(* Logix 5000 project; controller ARS14002_PLC vendor 1 type 14 code 218 rev 30.11; software revision 30.01; part 12 of 13 *)
(* tags used below, declared in another part *)
   AN_1000C : CM_AI_SCL;
   AN_200A : CM_AI_SCL;
   ARS_COLLECT : BOOL;
   ARS_FULL_COLLECTION : BOOL;
   ARS_FULL_COLLECTION_LATCH : BOOL;   // LATCHES THE FIRST TIME ARS HITS FULL COLLECTION DURING A MODE_ATOMIZE
   ARS_FULL_COLLECTION_TMR : TIMER;
   AT2_AtomizingStatus_OSF_OB : BOOL;
   AT2_FT_202_TOTAL_HEAT : REAL;
   AT2_HIBON_DISCHARGE_TEMP : REAL;
   AT2_HIBON_DISCHARGE_TEMP_MAX : REAL;
   AT2_PLANT_ATOMIZING : BOOL;
   AT2_PLANT_COLLECTION_PERCENT : REAL;
   AT2_PLANT_COLLECTION_PERCENT_GOOD_GAS : REAL;
   AT2_PLANT_COLLECTION_TIME : TIMER;
   AT2_PLANT_GOOD_GAS_PERCENT : REAL;
   AT2_PLANT_GOOD_GAS_TIME : TIMER;   // AT2 total time with good gas and no collection stops
   AT2_PLANT_GOOD_H2O_PERCENT : REAL;
   AT2_PLANT_GOOD_H2O_TIME : TIMER;   // AT2 time with good dew point and no collection stop
   AT2_PLANT_GOOD_O2_PERCENT : REAL;
   AT2_PLANT_GOOD_O2_TIME : TIMER;   // AT2 time with good O2 and no collection stop
   AT2_PLANT_LIKELY_COLLECTION_TIME : TIMER;
   AT2_PLANT_MAX_H2O : REAL;
   AT2_PLANT_MAX_O2 : REAL;
   AT2_PLANT_POST_HEAT_NOTIFICATION_TON : TIMER;
   AT2_V1_OPEN : BOOL;
   AT2_V1_OPEN_OSR_OB : BOOL;
   AT2_V1_OPEN_OSR_SB : BOOL;
   AT2_V1_OPEN_POSTHEAT_CTR : COUNTER;
   AT3_AtomizingStatus_OSF_OB : BOOL;
   AT3_FT_202_TOTAL_HEAT : REAL;
   AT3_HIBON_DISCHARGE_TEMP : REAL;
   AT3_HIBON_DISCHARGE_TEMP_MAX : REAL;
   AT3_PLANT_ATOMIZING : BOOL;
   AT3_PLANT_COLLECTION_PERCENT : REAL;
   AT3_PLANT_COLLECTION_PERCENT_GOOD_GAS : REAL;
   AT3_PLANT_COLLECTION_TIME : TIMER;
   AT3_PLANT_GOOD_GAS_PERCENT : REAL;
   AT3_PLANT_GOOD_GAS_TIME : TIMER;   // total time with good gas and no collection stops
   AT3_PLANT_GOOD_H2O_PERCENT : REAL;
   AT3_PLANT_GOOD_H2O_TIME : TIMER;   // time with good dew point and no collection stop
   AT3_PLANT_GOOD_O2_PERCENT : REAL;
   AT3_PLANT_GOOD_O2_TIME : TIMER;   // time with good O2 and no collection stop
   AT3_PLANT_LIKELY_COLLECTION_TIME : TIMER;
   AT3_PLANT_MAX_H2O : REAL;
   AT3_PLANT_MAX_O2 : REAL;
   AT3_PLANT_POST_HEAT_NOTIFICATION_TON : TIMER;
   AT3_V1_OPEN : BOOL;
   AT3_V1_OPEN_OSR_OB : BOOL;
   AT3_V1_OPEN_OSR_SB : BOOL;
   AT3_V1_OPEN_POSTHEAT_CTR : COUNTER;
   CALC_FT_1002_MONTH_RETURN : REAL;
   CALC_FT_1002_MONTH_TOTALIZER_RESET : BOOL;
   CALC_FT_1002_MONTH_TOTALIZER_START : BOOL;
   CALC_FT_1002_MONTH_TOTALIZER_STOP : BOOL;
   CALC_FT_1002_TOTAL_RETURN : REAL;
   CALC_FT_202_MONTH : REAL;
   CALC_FT_202_TOTAL_HEAT : REAL;
   CALC_NEXT_DAY_OSR_OB : BOOL;
   CALC_NEXT_MONTH_OSR_OB : BOOL;
   COLDBOX_REACTION_TMR : TIMER;
   COLDBOX_REACTION_TMR_SEC : REAL;
   FCV_1001 : CM_AO_VLV;
   FCV_1002 : CM_AO_VLV;
   FCV_101A : CM_AO_VLV;
   FCV_101A_ZT_OSR : BOOL;
   FCV_101B : CM_AO_VLV;
   FCV_101B_ZT_OSR : BOOL;
   FCV_101C : CM_AO_VLV;
   FCV_101C_ZT_OSR : BOOL;
   FCV_102A : CM_AO_VLV;
   FCV_102A_COLLECTION_CV_HIGH : REAL;
   FCV_102B : CM_AO_VLV;
   FCV_102B_COLLECTION_CV_HIGH : REAL;
   FCV_102C : CM_AO_VLV;
   FCV_102C_COLLECTION_CV_HIGH : REAL;
   FCV_1221 : CM_AO_VLV;
   FCV_1251 : CM_AO_VLV;
   FCV_202 : CM_AO_VLV;
   FCV_202_COLLECTION_CV_LOW : REAL;
   FCV_202_HEAT_AVG : REAL;
   FCV_202_HEAT_AVG_TON : TIMER;
   FCV_202_HEAT_TOTAL : REAL;
   FCV_202_SAMPLES : COUNTER;
   FCV_204 : CM_AO_VLV;
   FCV_204_COLLECTION_CV_HIGH : REAL;
   FCV_204_HEAT_AVG : REAL;
   FCV_204_HEAT_TOTAL : REAL;
   FCV_207 : CM_AO_VLV;
   FCV_504 : CM_AO_VLV;
   FCV_603 : CM_AO_VLV;
   FCV_605 : CM_AO_VLV;
   FCV_753 : CM_AO_VLV;
   FCV_754 : CM_AO_VLV;
   FCV_755 : CM_AO_VLV;
   FT_1002 : CM_AI_SCL;
   FT_202_ALT_SCFM : REAL;
   FULL_COLLECT_INTERRUPT_ALM : BOOL;
   FULL_COLLECT_INTERRUPT_ALM_TIME : DINT;
   FULL_COLLECT_INTERRUPT_ALM_TMR : TIMER;
   FULL_COLLECT_START_ALM : BOOL;
   FULL_COLLECT_START_ALM_TIME : DINT;
   FULL_COLLECT_START_ALM_TMR : TIMER;
   Heat_Counter_AT2 : DINT;
   Heat_Counter_AT3 : REAL;
   Heat_Counter_Month : REAL;
   Heat_Counter_Pilot : REAL;
   HEAT_TIMER_AT2 : TIMER;
   HEAT_TIMER_AT3 : TIMER;
   MODE_ATOMIZE : BOOL;
   P_800A_CAVIT_CTR_MONTH : COUNTER;
   P_800B_CAVIT_CTR_MONTH : COUNTER;
   P_800C_CAVIT_CTR_MONTH : COUNTER;
   P_800D_CAVIT_CTR_MONTH : COUNTER;
   Pilot_AtomizingStatus_OSF_OB : BOOL;
   PILOT_FT_202_TOTAL_HEAT : REAL;
   PILOT_PLANT_ATOMIZING : BOOL;
   PILOT_PLANT_MAX_H2O : REAL;
   PILOT_PLANT_MAX_O2 : REAL;
   PILOT_PLANT_POST_HEAT_NOTIFICATION_TON : TIMER;
   PWHMI_AtomizingStatus_OSR_OB : BOOL;
   SEND_AT2_PLANT_NOTICE : BOOL;
   SEND_AT3_PLANT_NOTICE : BOOL;
   SEND_PILOT_PLANT_NOTICE : BOOL;
   SV_202F : CM_DO_GENERIC;
   SV_802AX : CM_DO_GENERIC;
   SV_802AX_ONS : BOOL;
   SV_802BX : CM_DO_GENERIC;
   SV_802BX_ONS : BOOL;
   SV_802CX : CM_DO_GENERIC;
   SV_802CX_ONS : BOOL;
   SV_802DX : CM_DO_GENERIC;
   SV_802DX_ONS : BOOL;
   XV_802_VENT_COUNTER : COUNTER;
   XV_802_VENT_TOTAL_TIME : TIMER;
   ZT_1001 : CM_AI_SCL;
   ZT_1002 : CM_AI_SCL;
   ZT_101A : CM_AI_SCL;
   ZT_101B : CM_AI_SCL;
   ZT_101C : CM_AI_SCL;
   ZT_102A : CM_AI_SCL;
   ZT_102B : CM_AI_SCL;
   ZT_102C : CM_AI_SCL;
   ZT_1221 : CM_AI_SCL;
   ZT_1251 : CM_AI_SCL;
   ZT_202 : CM_AI_SCL;
   ZT_204 : CM_AI_SCL;
   ZT_207 : CM_AI_SCL;
   ZT_504 : CM_AI_SCL;
   ZT_603 : CM_AI_SCL;
   ZT_605 : CM_AI_SCL;
   ZT_753 : CM_AI_SCL;
   ZT_754 : CM_AI_SCL;
   ZT_755 : CM_AI_SCL;
(* MainProgram, continued *)

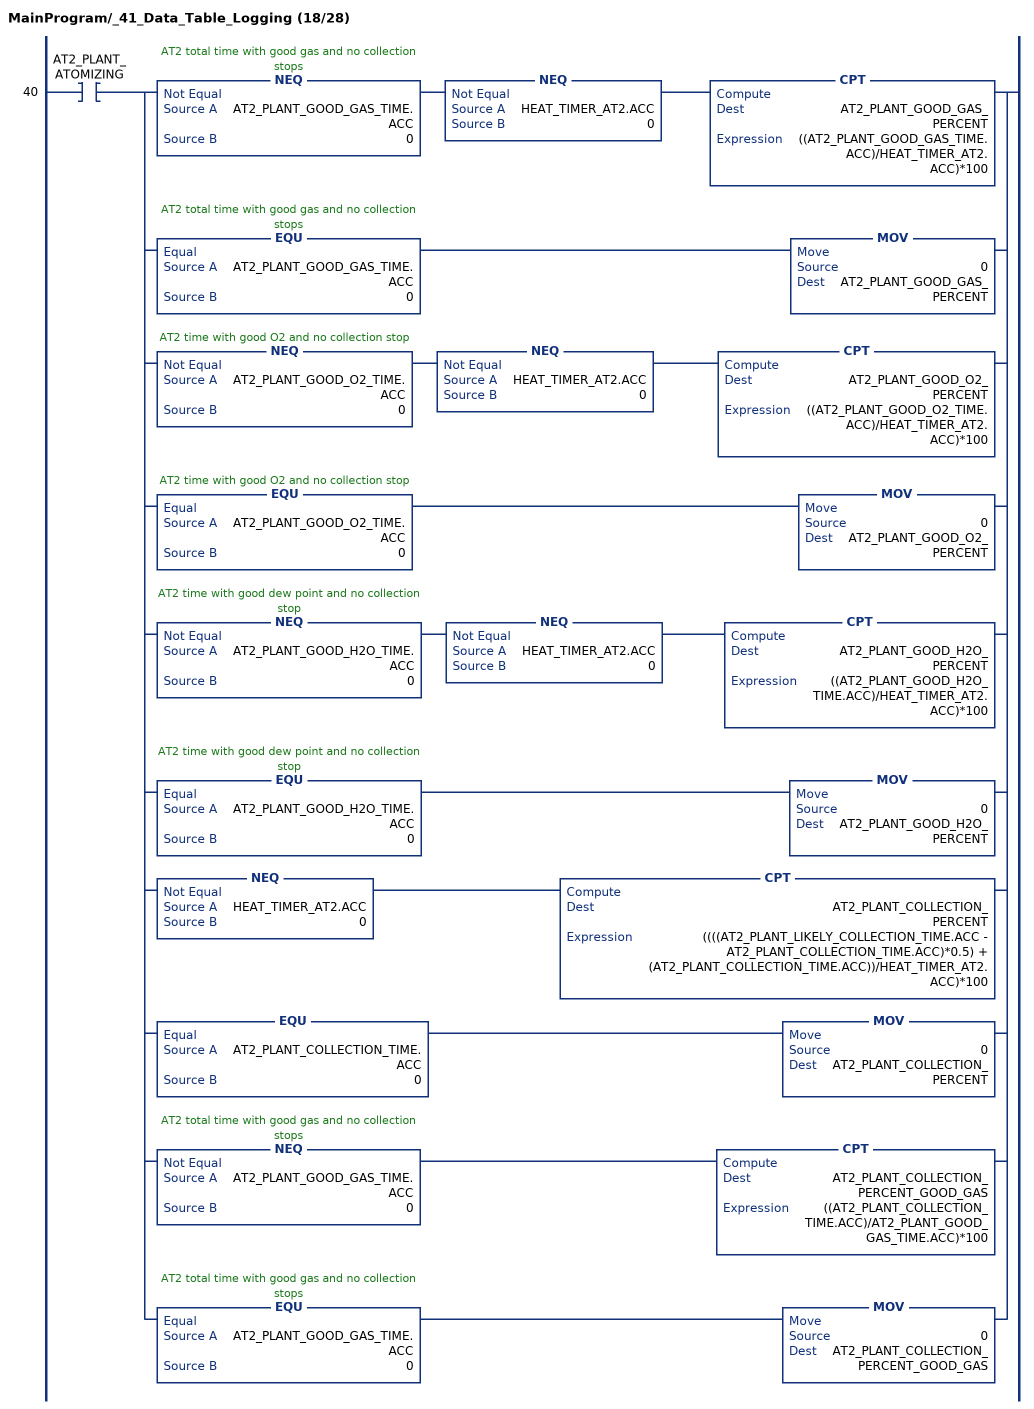
   [picture p246: MainProgram/_41_Data_Table_Logging rungs 40-40]
   40: XIC(AT2_PLANT_ATOMIZING)[NEQ(AT2_PLANT_GOOD_GAS_TIME.ACC,0) NEQ(HEAT_TIMER_AT2.ACC,0) CPT(AT2_PLANT_GOOD_GAS_PERCENT,((AT2_PLANT_GOOD_GAS_TIME.ACC)/HEAT_TIMER_AT2.ACC)*100) ,EQU(AT2_PLANT_GOOD_GAS_TIME.ACC,0) MOV(0,AT2_PLANT_GOOD_GAS_PERCENT) ,NEQ(AT2_PLANT_GOOD_O2_TIME.ACC,0) NEQ(HEAT_TIMER_AT2.ACC,0) CPT(AT2_PLANT_GOOD_O2_PERCENT,((AT2_PLANT_GOOD_O2_TIME.ACC)/HEAT_TIMER_AT2.ACC)*100) ,EQU(AT2_PLANT_GOOD_O2_TIME.ACC,0) MOV(0,AT2_PLANT_GOOD_O2_PERCENT) ,NEQ(AT2_PLANT_GOOD_H2O_TIME.ACC,0) NEQ(HEAT_TIMER_AT2.ACC,0) CPT(AT2_PLANT_GOOD_H2O_PERCENT,((AT2_PLANT_GOOD_H2O_TIME.ACC)/HEAT_TIMER_AT2.ACC)*100) ,EQU(AT2_PLANT_GOOD_H2O_TIME.ACC,0) MOV(0,AT2_PLANT_GOOD_H2O_PERCENT) ,NEQ(HEAT_TIMER_AT2.ACC,0) CPT(AT2_PLANT_COLLECTION_PERCENT,((((AT2_PLANT_LIKELY_COLLECTION_TIME.ACC - AT2_PLANT_COLLECTION_TIME.ACC)*0.5) + (AT2_PLANT_COLLECTION_TIME.ACC))/HEAT_TIMER_AT2.ACC)*100) ,EQU(AT2_PLANT_COLLECTION_TIME.ACC,0) MOV(0,AT2_PLANT_COLLECTION_PERCENT) ,NEQ(AT2_PLANT_GOOD_GAS_TIME.ACC,0) CPT(AT2_PLANT_COLLECTION_PERCENT_GOOD_GAS,((AT2_PLANT_COLLECTION_TIME.ACC)/AT2_PLANT_GOOD_GAS_TIME.ACC)*100) ,EQU(AT2_PLANT_GOOD_GAS_TIME.ACC,0) MOV(0,AT2_PLANT_COLLECTION_PERCENT_GOOD_GAS) ];
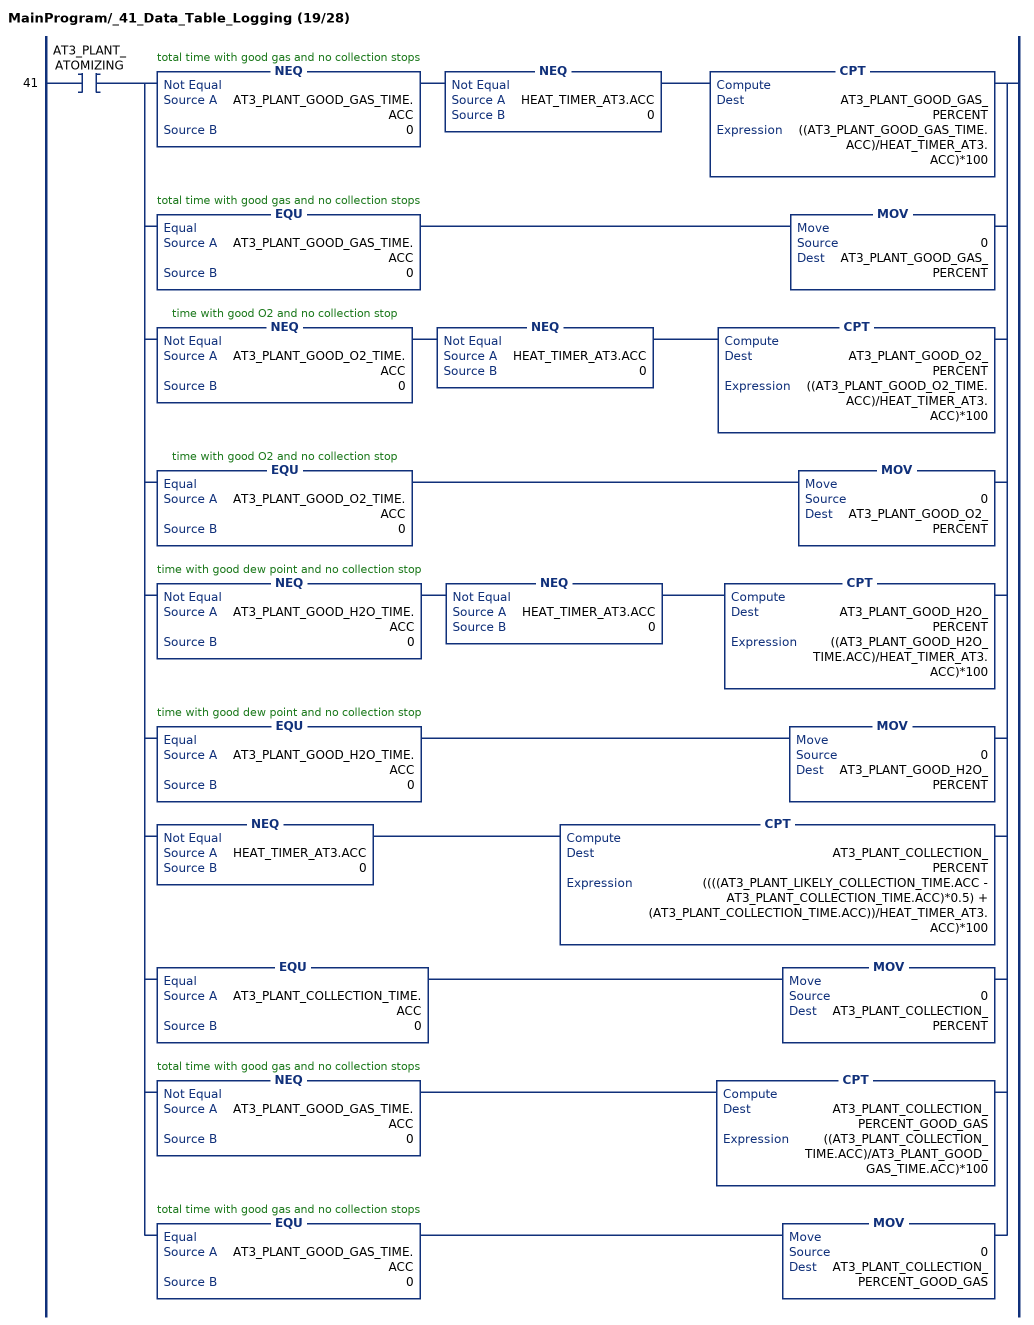
   41: XIC(AT3_PLANT_ATOMIZING)[NEQ(AT3_PLANT_GOOD_GAS_TIME.ACC,0) NEQ(HEAT_TIMER_AT3.ACC,0) CPT(AT3_PLANT_GOOD_GAS_PERCENT,((AT3_PLANT_GOOD_GAS_TIME.ACC)/HEAT_TIMER_AT3.ACC)*100) ,EQU(AT3_PLANT_GOOD_GAS_TIME.ACC,0) MOV(0,AT3_PLANT_GOOD_GAS_PERCENT) ,NEQ(AT3_PLANT_GOOD_O2_TIME.ACC,0) NEQ(HEAT_TIMER_AT3.ACC,0) CPT(AT3_PLANT_GOOD_O2_PERCENT,((AT3_PLANT_GOOD_O2_TIME.ACC)/HEAT_TIMER_AT3.ACC)*100) ,EQU(AT3_PLANT_GOOD_O2_TIME.ACC,0) MOV(0,AT3_PLANT_GOOD_O2_PERCENT) ,NEQ(AT3_PLANT_GOOD_H2O_TIME.ACC,0) NEQ(HEAT_TIMER_AT3.ACC,0) CPT(AT3_PLANT_GOOD_H2O_PERCENT,((AT3_PLANT_GOOD_H2O_TIME.ACC)/HEAT_TIMER_AT3.ACC)*100) ,EQU(AT3_PLANT_GOOD_H2O_TIME.ACC,0) MOV(0,AT3_PLANT_GOOD_H2O_PERCENT) ,NEQ(HEAT_TIMER_AT3.ACC,0) CPT(AT3_PLANT_COLLECTION_PERCENT,((((AT3_PLANT_LIKELY_COLLECTION_TIME.ACC - AT3_PLANT_COLLECTION_TIME.ACC)*0.5) + (AT3_PLANT_COLLECTION_TIME.ACC))/HEAT_TIMER_AT3.ACC)*100) ,EQU(AT3_PLANT_COLLECTION_TIME.ACC,0) MOV(0,AT3_PLANT_COLLECTION_PERCENT) ,NEQ(AT3_PLANT_GOOD_GAS_TIME.ACC,0) CPT(AT3_PLANT_COLLECTION_PERCENT_GOOD_GAS,((AT3_PLANT_COLLECTION_TIME.ACC)/AT3_PLANT_GOOD_GAS_TIME.ACC)*100) ,EQU(AT3_PLANT_GOOD_GAS_TIME.ACC,0) MOV(0,AT3_PLANT_COLLECTION_PERCENT_GOOD_GAS) ];
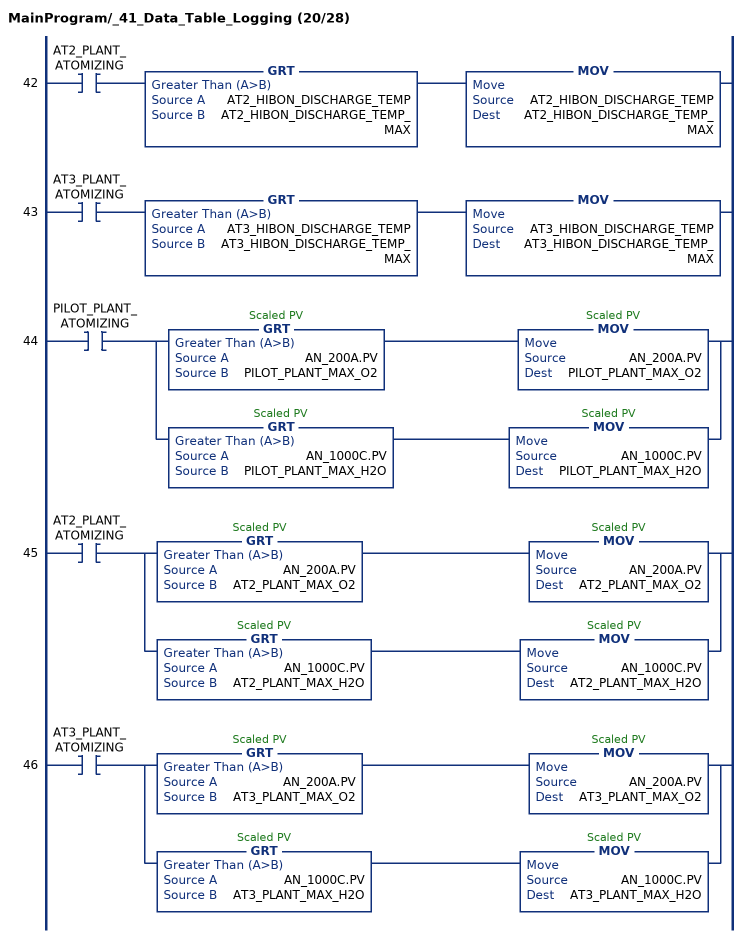
   42: XIC(AT2_PLANT_ATOMIZING)GRT(AT2_HIBON_DISCHARGE_TEMP,AT2_HIBON_DISCHARGE_TEMP_MAX)MOV(AT2_HIBON_DISCHARGE_TEMP,AT2_HIBON_DISCHARGE_TEMP_MAX);
   43: XIC(AT3_PLANT_ATOMIZING)GRT(AT3_HIBON_DISCHARGE_TEMP,AT3_HIBON_DISCHARGE_TEMP_MAX)MOV(AT3_HIBON_DISCHARGE_TEMP,AT3_HIBON_DISCHARGE_TEMP_MAX);
   44: XIC(PILOT_PLANT_ATOMIZING)[GRT(AN_200A.PV,PILOT_PLANT_MAX_O2) MOV(AN_200A.PV,PILOT_PLANT_MAX_O2) ,GRT(AN_1000C.PV,PILOT_PLANT_MAX_H2O) MOV(AN_1000C.PV,PILOT_PLANT_MAX_H2O) ];
   45: XIC(AT2_PLANT_ATOMIZING)[GRT(AN_200A.PV,AT2_PLANT_MAX_O2) MOV(AN_200A.PV,AT2_PLANT_MAX_O2) ,GRT(AN_1000C.PV,AT2_PLANT_MAX_H2O) MOV(AN_1000C.PV,AT2_PLANT_MAX_H2O) ];
   46: XIC(AT3_PLANT_ATOMIZING)[GRT(AN_200A.PV,AT3_PLANT_MAX_O2) MOV(AN_200A.PV,AT3_PLANT_MAX_O2) ,GRT(AN_1000C.PV,AT3_PLANT_MAX_H2O) MOV(AN_1000C.PV,AT3_PLANT_MAX_H2O) ];
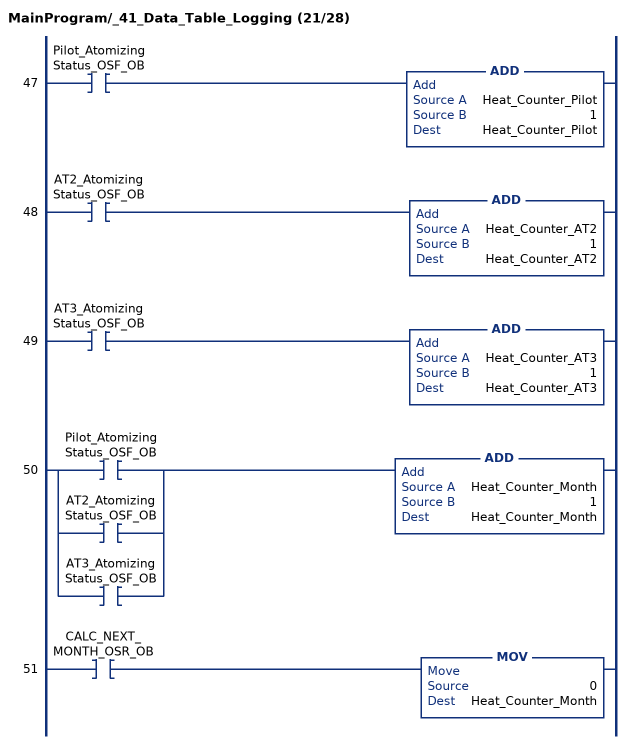
   47: XIC(Pilot_AtomizingStatus_OSF_OB)ADD(Heat_Counter_Pilot,1,Heat_Counter_Pilot);
   48: XIC(AT2_AtomizingStatus_OSF_OB)ADD(Heat_Counter_AT2,1,Heat_Counter_AT2);
   49: XIC(AT3_AtomizingStatus_OSF_OB)ADD(Heat_Counter_AT3,1,Heat_Counter_AT3);
   50: [XIC(Pilot_AtomizingStatus_OSF_OB) ,XIC(AT2_AtomizingStatus_OSF_OB) ,XIC(AT3_AtomizingStatus_OSF_OB) ]ADD(Heat_Counter_Month,1,Heat_Counter_Month);
   51: XIC(CALC_NEXT_MONTH_OSR_OB)MOV(0,Heat_Counter_Month);
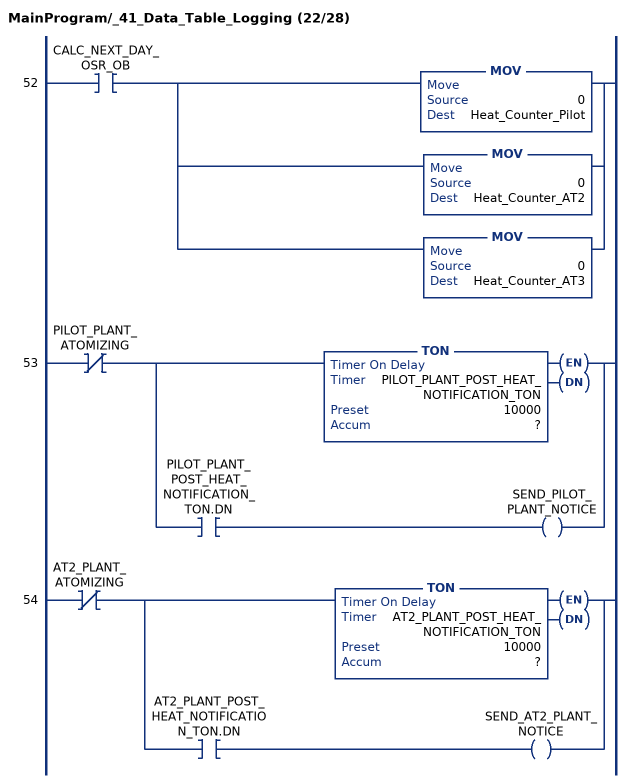
   52: XIC(CALC_NEXT_DAY_OSR_OB)[MOV(0,Heat_Counter_Pilot) ,MOV(0,Heat_Counter_AT2) ,MOV(0,Heat_Counter_AT3) ];
   53: XIO(PILOT_PLANT_ATOMIZING)[TON(PILOT_PLANT_POST_HEAT_NOTIFICATION_TON,?,?) ,XIC(PILOT_PLANT_POST_HEAT_NOTIFICATION_TON.DN) OTE(SEND_PILOT_PLANT_NOTICE) ];
   54: XIO(AT2_PLANT_ATOMIZING)[TON(AT2_PLANT_POST_HEAT_NOTIFICATION_TON,?,?) ,XIC(AT2_PLANT_POST_HEAT_NOTIFICATION_TON.DN) OTE(SEND_AT2_PLANT_NOTICE) ];
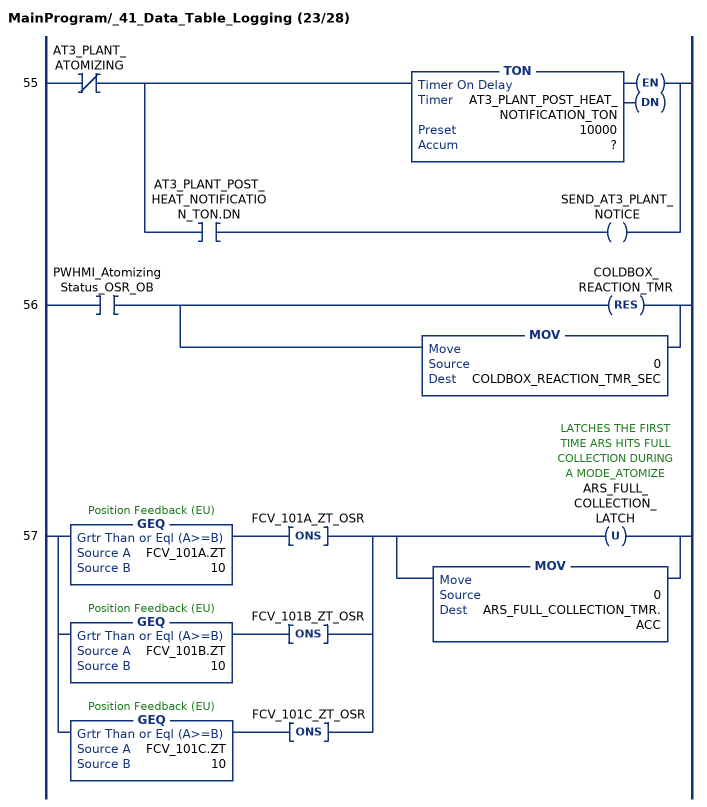
   55: XIO(AT3_PLANT_ATOMIZING)[TON(AT3_PLANT_POST_HEAT_NOTIFICATION_TON,?,?) ,XIC(AT3_PLANT_POST_HEAT_NOTIFICATION_TON.DN) OTE(SEND_AT3_PLANT_NOTICE) ];
   56: XIC(PWHMI_AtomizingStatus_OSR_OB)[RES(COLDBOX_REACTION_TMR) ,MOV(0,COLDBOX_REACTION_TMR_SEC) ];
   57: [GEQ(FCV_101A.ZT,10) ONS(FCV_101A_ZT_OSR) ,GEQ(FCV_101B.ZT,10) ONS(FCV_101B_ZT_OSR) ,GEQ(FCV_101C.ZT,10) ONS(FCV_101C_ZT_OSR) ][OTU(ARS_FULL_COLLECTION_LATCH) ,MOV(0,ARS_FULL_COLLECTION_TMR.ACC) ];
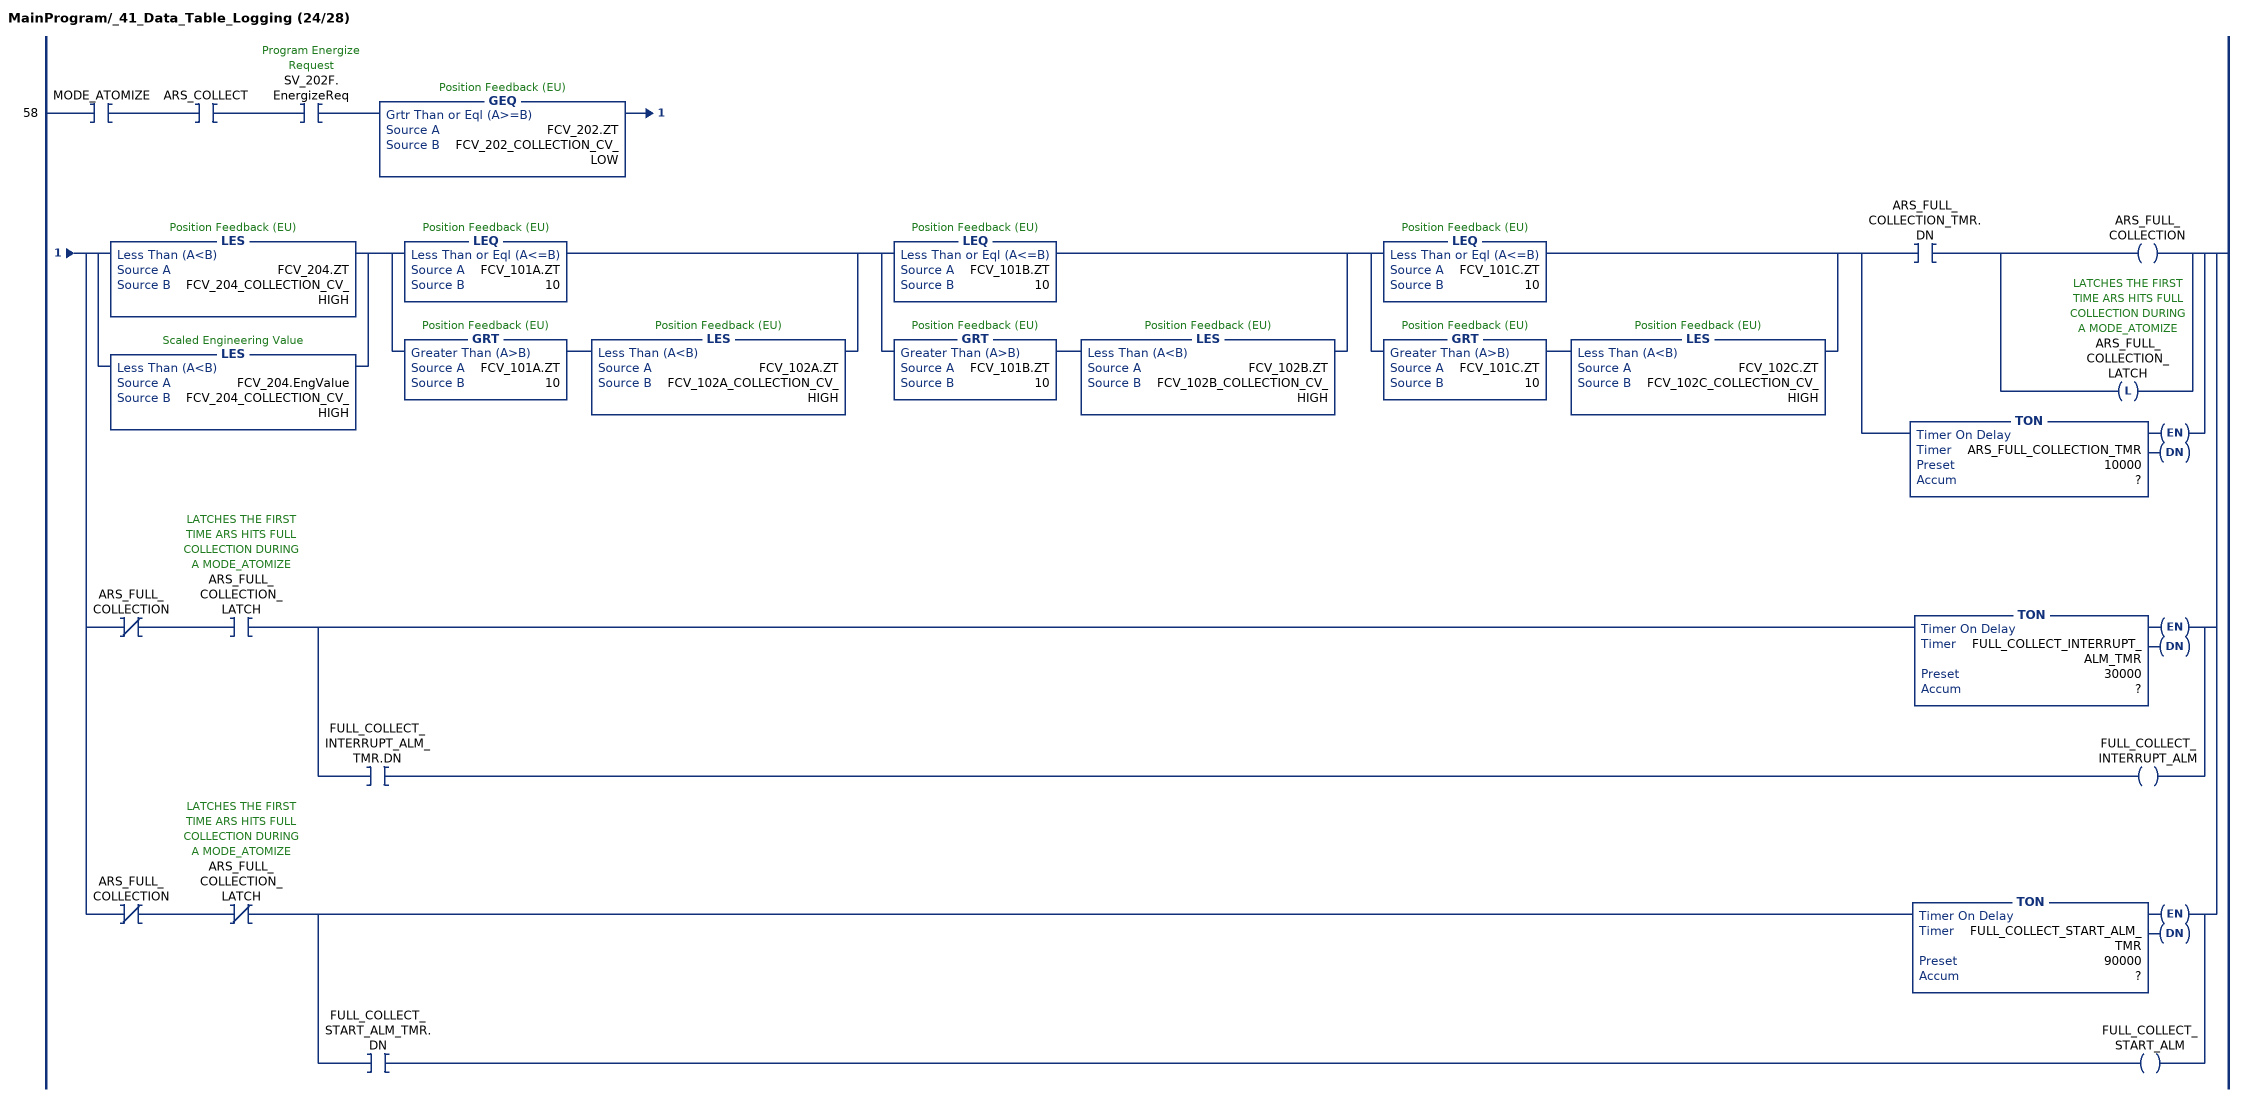
   58: XIC(MODE_ATOMIZE)XIC(ARS_COLLECT)XIC(SV_202F.EnergizeReq)GEQ(FCV_202.ZT,FCV_202_COLLECTION_CV_LOW)[[LES(FCV_204.ZT,FCV_204_COLLECTION_CV_HIGH) ,LES(FCV_204.EngValue,FCV_204_COLLECTION_CV_HIGH) ] [LEQ(FCV_101A.ZT,10) ,GRT(FCV_101A.ZT,10) LES(FCV_102A.ZT,FCV_102A_COLLECTION_CV_HIGH) ] [LEQ(FCV_101B.ZT,10) ,GRT(FCV_101B.ZT,10) LES(FCV_102B.ZT,FCV_102B_COLLECTION_CV_HIGH) ] [LEQ(FCV_101C.ZT,10) ,GRT(FCV_101C.ZT,10) LES(FCV_102C.ZT,FCV_102C_COLLECTION_CV_HIGH) ] [XIC(ARS_FULL_COLLECTION_TMR.DN) [OTE(ARS_FULL_COLLECTION) ,OTL(ARS_FULL_COLLECTION_LATCH) ] ,TON(ARS_FULL_COLLECTION_TMR,?,?) ] ,XIO(ARS_FULL_COLLECTION) XIC(ARS_FULL_COLLECTION_LATCH) [TON(FULL_COLLECT_INTERRUPT_ALM_TMR,?,?) ,XIC(FULL_COLLECT_INTERRUPT_ALM_TMR.DN) OTE(FULL_COLLECT_INTERRUPT_ALM) ] ,XIO(ARS_FULL_COLLECTION) XIO(ARS_FULL_COLLECTION_LATCH) [TON(FULL_COLLECT_START_ALM_TMR,?,?) ,XIC(FULL_COLLECT_START_ALM_TMR.DN) OTE(FULL_COLLECT_START_ALM) ] ];
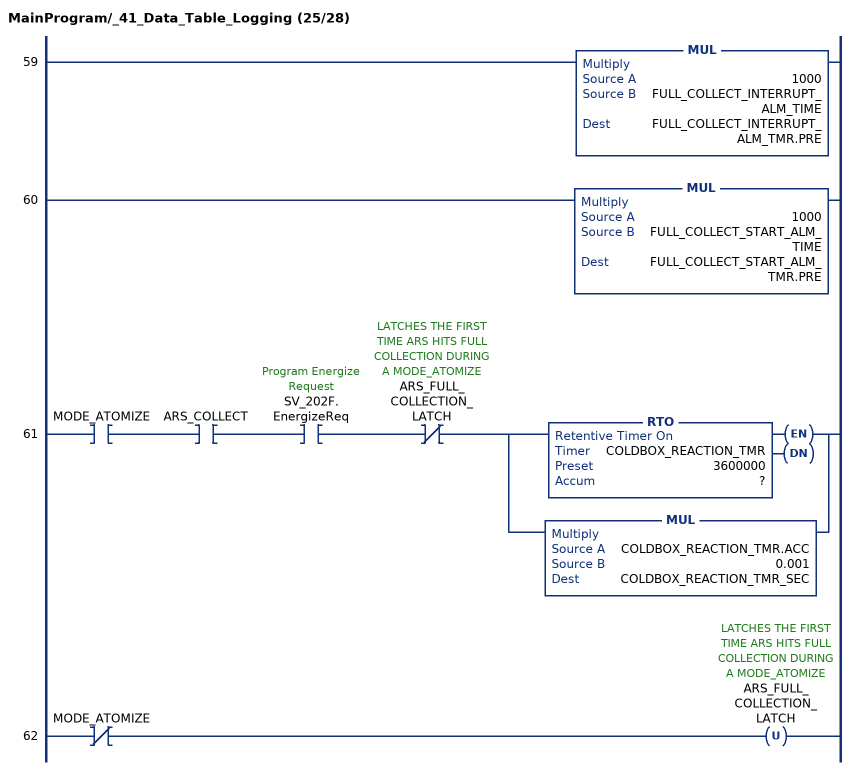
   59: MUL(1000,FULL_COLLECT_INTERRUPT_ALM_TIME,FULL_COLLECT_INTERRUPT_ALM_TMR.PRE);
   60: MUL(1000,FULL_COLLECT_START_ALM_TIME,FULL_COLLECT_START_ALM_TMR.PRE);
   61: XIC(MODE_ATOMIZE)XIC(ARS_COLLECT)XIC(SV_202F.EnergizeReq)XIO(ARS_FULL_COLLECTION_LATCH)[RTO(COLDBOX_REACTION_TMR,?,?) ,MUL(COLDBOX_REACTION_TMR.ACC,0.001,COLDBOX_REACTION_TMR_SEC) ];
   62: XIO(MODE_ATOMIZE)OTU(ARS_FULL_COLLECTION_LATCH);
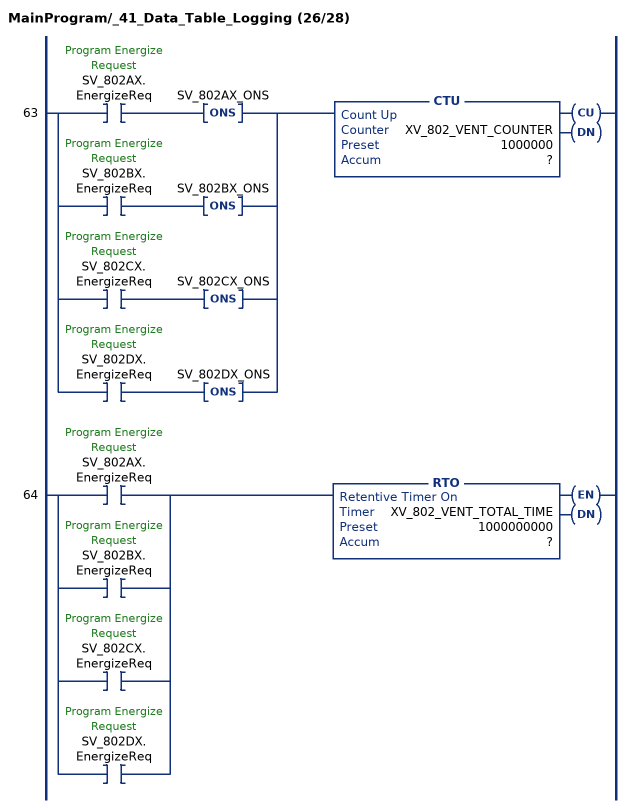
   63: [XIC(SV_802AX.EnergizeReq) ONS(SV_802AX_ONS) ,XIC(SV_802BX.EnergizeReq) ONS(SV_802BX_ONS) ,XIC(SV_802CX.EnergizeReq) ONS(SV_802CX_ONS) ,XIC(SV_802DX.EnergizeReq) ONS(SV_802DX_ONS) ]CTU(XV_802_VENT_COUNTER,?,?);
   64: [XIC(SV_802AX.EnergizeReq) ,XIC(SV_802BX.EnergizeReq) ,XIC(SV_802CX.EnergizeReq) ,XIC(SV_802DX.EnergizeReq) ]RTO(XV_802_VENT_TOTAL_TIME,?,?);
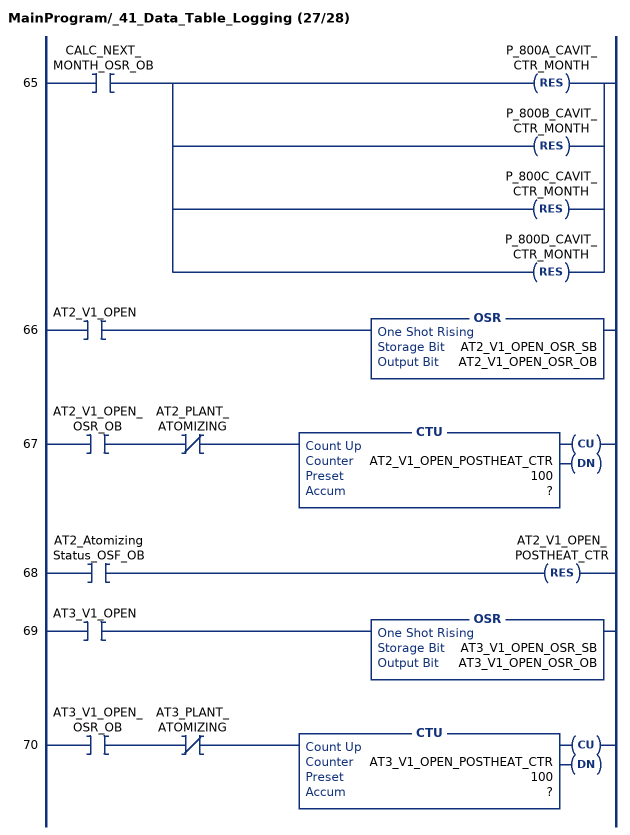
   65: XIC(CALC_NEXT_MONTH_OSR_OB)[RES(P_800A_CAVIT_CTR_MONTH) ,RES(P_800B_CAVIT_CTR_MONTH) ,RES(P_800C_CAVIT_CTR_MONTH) ,RES(P_800D_CAVIT_CTR_MONTH) ];
   66: XIC(AT2_V1_OPEN)OSR(AT2_V1_OPEN_OSR_SB,AT2_V1_OPEN_OSR_OB);
   67: XIC(AT2_V1_OPEN_OSR_OB)XIO(AT2_PLANT_ATOMIZING)CTU(AT2_V1_OPEN_POSTHEAT_CTR,?,?);
   68: XIC(AT2_AtomizingStatus_OSF_OB)RES(AT2_V1_OPEN_POSTHEAT_CTR);
   69: XIC(AT3_V1_OPEN)OSR(AT3_V1_OPEN_OSR_SB,AT3_V1_OPEN_OSR_OB);
   70: XIC(AT3_V1_OPEN_OSR_OB)XIO(AT3_PLANT_ATOMIZING)CTU(AT3_V1_OPEN_POSTHEAT_CTR,?,?);
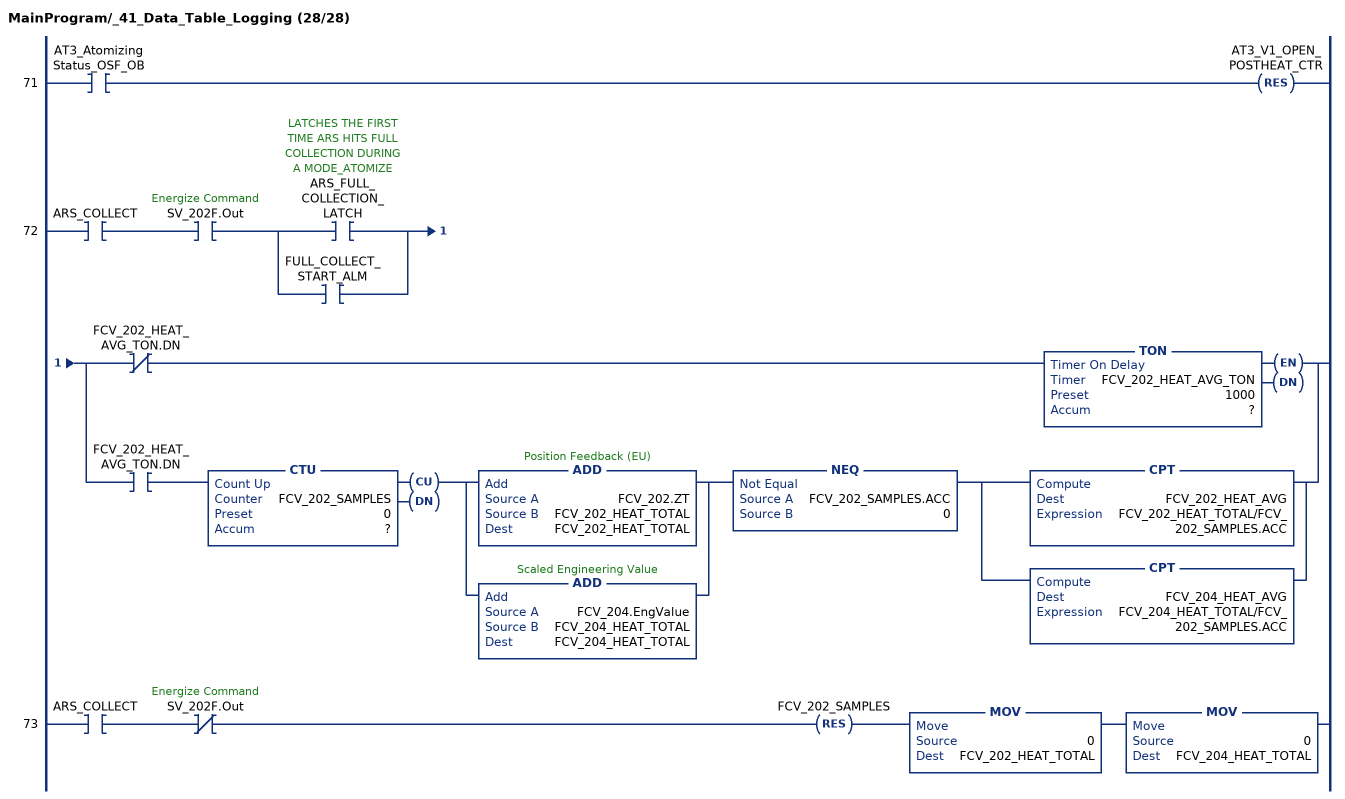
   71: XIC(AT3_AtomizingStatus_OSF_OB)RES(AT3_V1_OPEN_POSTHEAT_CTR);
   72: XIC(ARS_COLLECT)XIC(SV_202F.Out)[XIC(ARS_FULL_COLLECTION_LATCH) ,XIC(FULL_COLLECT_START_ALM) ][XIO(FCV_202_HEAT_AVG_TON.DN) TON(FCV_202_HEAT_AVG_TON,?,?) ,XIC(FCV_202_HEAT_AVG_TON.DN) CTU(FCV_202_SAMPLES,?,?) [ADD(FCV_202.ZT,FCV_202_HEAT_TOTAL,FCV_202_HEAT_TOTAL) ,ADD(FCV_204.EngValue,FCV_204_HEAT_TOTAL,FCV_204_HEAT_TOTAL) ] NEQ(FCV_202_SAMPLES.ACC,0) [CPT(FCV_202_HEAT_AVG,FCV_202_HEAT_TOTAL/FCV_202_SAMPLES.ACC) ,CPT(FCV_204_HEAT_AVG,FCV_204_HEAT_TOTAL/FCV_202_SAMPLES.ACC) ] ];
   73: XIC(ARS_COLLECT)XIO(SV_202F.Out)RES(FCV_202_SAMPLES)MOV(0,FCV_202_HEAT_TOTAL)MOV(0,FCV_204_HEAT_TOTAL);
END_ROUTINE

ROUTINE _42_Flow_Totalizer   (* function block diagram *)
   SHEET 1
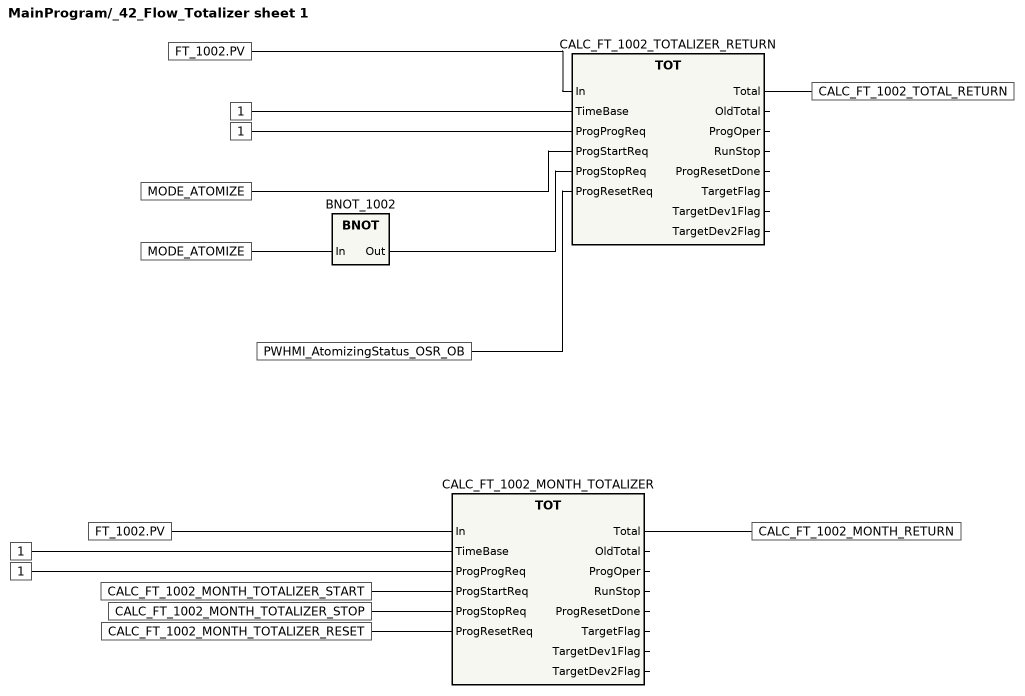
   BNOT_1002 : BNOT(In := MODE_ATOMIZE);
   CALC_FT_1002_MONTH_TOTALIZER : TOT(In := FT_1002.PV, TimeBase := 1, ProgProgReq := 1, ProgStartReq := CALC_FT_1002_MONTH_TOTALIZER_START, ProgStopReq := CALC_FT_1002_MONTH_TOTALIZER_STOP, ProgResetReq := CALC_FT_1002_MONTH_TOTALIZER_RESET);   // unwired pins: OldTotal ProgOper RunStop ProgResetDone TargetFlag TargetDev1Flag TargetDev2Flag
   CALC_FT_1002_TOTALIZER_RETURN : TOT(In := FT_1002.PV, TimeBase := 1, ProgProgReq := 1, ProgStartReq := MODE_ATOMIZE, ProgStopReq := BNOT_1002.Out, ProgResetReq := PWHMI_AtomizingStatus_OSR_OB);   // unwired pins: OldTotal ProgOper RunStop ProgResetDone TargetFlag TargetDev1Flag TargetDev2Flag
   CALC_FT_1002_MONTH_RETURN := CALC_FT_1002_MONTH_TOTALIZER.Total;
   CALC_FT_1002_TOTAL_RETURN := CALC_FT_1002_TOTALIZER_RETURN.Total;
   SHEET 2
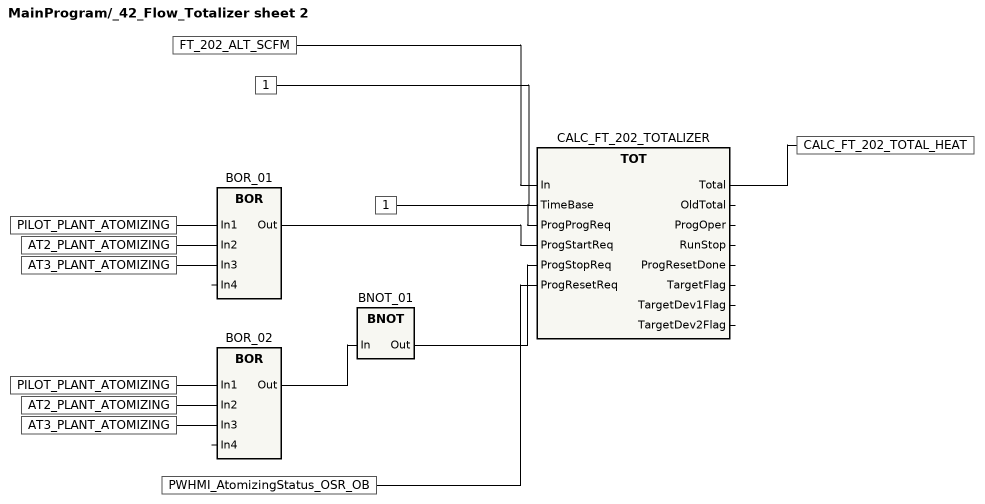
   BOR_01 : BOR(In1 := PILOT_PLANT_ATOMIZING, In2 := AT2_PLANT_ATOMIZING, In3 := AT3_PLANT_ATOMIZING);   // unwired pins: In4
   BOR_02 : BOR(In1 := PILOT_PLANT_ATOMIZING, In2 := AT2_PLANT_ATOMIZING, In3 := AT3_PLANT_ATOMIZING);   // unwired pins: In4
   BNOT_01 : BNOT(In := BOR_02.Out);
   CALC_FT_202_TOTALIZER : TOT(In := FT_202_ALT_SCFM, TimeBase := 1, ProgProgReq := 1, ProgStartReq := BOR_01.Out, ProgStopReq := BNOT_01.Out, ProgResetReq := PWHMI_AtomizingStatus_OSR_OB);   // unwired pins: OldTotal ProgOper RunStop ProgResetDone TargetFlag TargetDev1Flag TargetDev2Flag
   CALC_FT_202_TOTAL_HEAT := CALC_FT_202_TOTALIZER.Total;
   SHEET 3
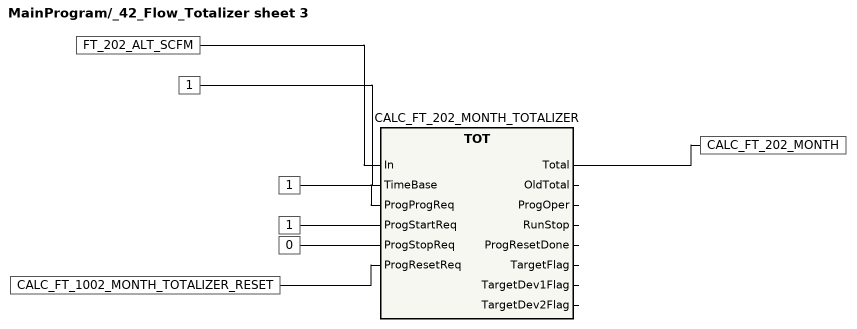
   CALC_FT_202_MONTH_TOTALIZER : TOT(In := FT_202_ALT_SCFM, TimeBase := 1, ProgProgReq := 1, ProgStartReq := 1, ProgStopReq := 0, ProgResetReq := CALC_FT_1002_MONTH_TOTALIZER_RESET);   // unwired pins: OldTotal ProgOper RunStop ProgResetDone TargetFlag TargetDev1Flag TargetDev2Flag
   CALC_FT_202_MONTH := CALC_FT_202_MONTH_TOTALIZER.Total;
   SHEET 4
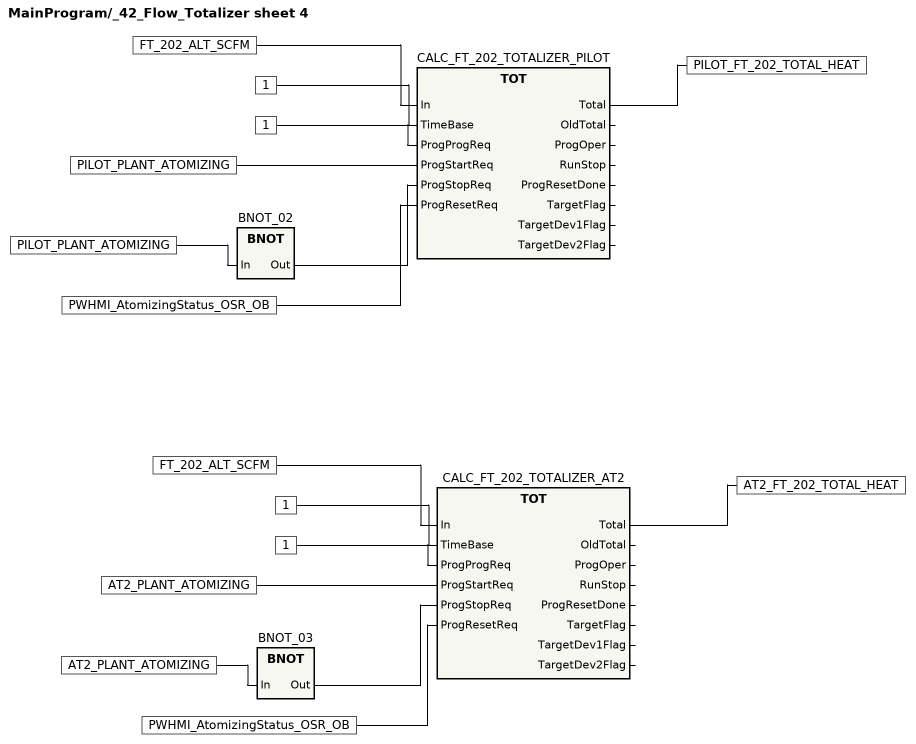
   BNOT_02 : BNOT(In := PILOT_PLANT_ATOMIZING);
   BNOT_03 : BNOT(In := AT2_PLANT_ATOMIZING);
   CALC_FT_202_TOTALIZER_PILOT : TOT(In := FT_202_ALT_SCFM, TimeBase := 1, ProgProgReq := 1, ProgStartReq := PILOT_PLANT_ATOMIZING, ProgStopReq := BNOT_02.Out, ProgResetReq := PWHMI_AtomizingStatus_OSR_OB);   // unwired pins: OldTotal ProgOper RunStop ProgResetDone TargetFlag TargetDev1Flag TargetDev2Flag
   CALC_FT_202_TOTALIZER_AT2 : TOT(In := FT_202_ALT_SCFM, TimeBase := 1, ProgProgReq := 1, ProgStartReq := AT2_PLANT_ATOMIZING, ProgStopReq := BNOT_03.Out, ProgResetReq := PWHMI_AtomizingStatus_OSR_OB);   // unwired pins: OldTotal ProgOper RunStop ProgResetDone TargetFlag TargetDev1Flag TargetDev2Flag
   PILOT_FT_202_TOTAL_HEAT := CALC_FT_202_TOTALIZER_PILOT.Total;
   AT2_FT_202_TOTAL_HEAT := CALC_FT_202_TOTALIZER_AT2.Total;
   SHEET 5
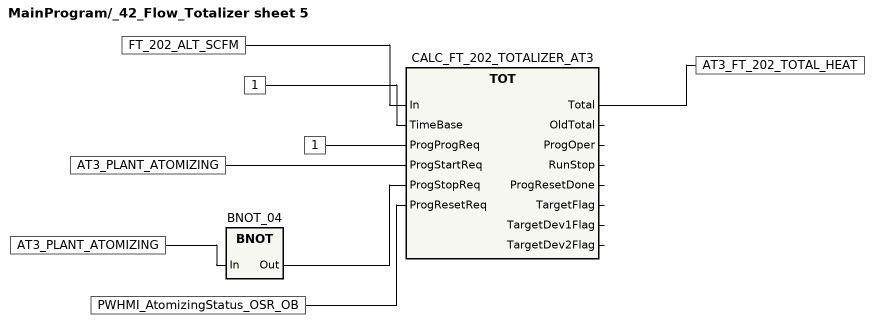
   BNOT_04 : BNOT(In := AT3_PLANT_ATOMIZING);
   CALC_FT_202_TOTALIZER_AT3 : TOT(In := FT_202_ALT_SCFM, TimeBase := 1, ProgProgReq := 1, ProgStartReq := AT3_PLANT_ATOMIZING, ProgStopReq := BNOT_04.Out, ProgResetReq := PWHMI_AtomizingStatus_OSR_OB);   // unwired pins: OldTotal ProgOper RunStop ProgResetDone TargetFlag TargetDev1Flag TargetDev2Flag
   AT3_FT_202_TOTAL_HEAT := CALC_FT_202_TOTALIZER_AT3.Total;
END_ROUTINE

ROUTINE _50_Outputs_Analog   (* ladder *)
// Analog Output scaling and alarm handling routine
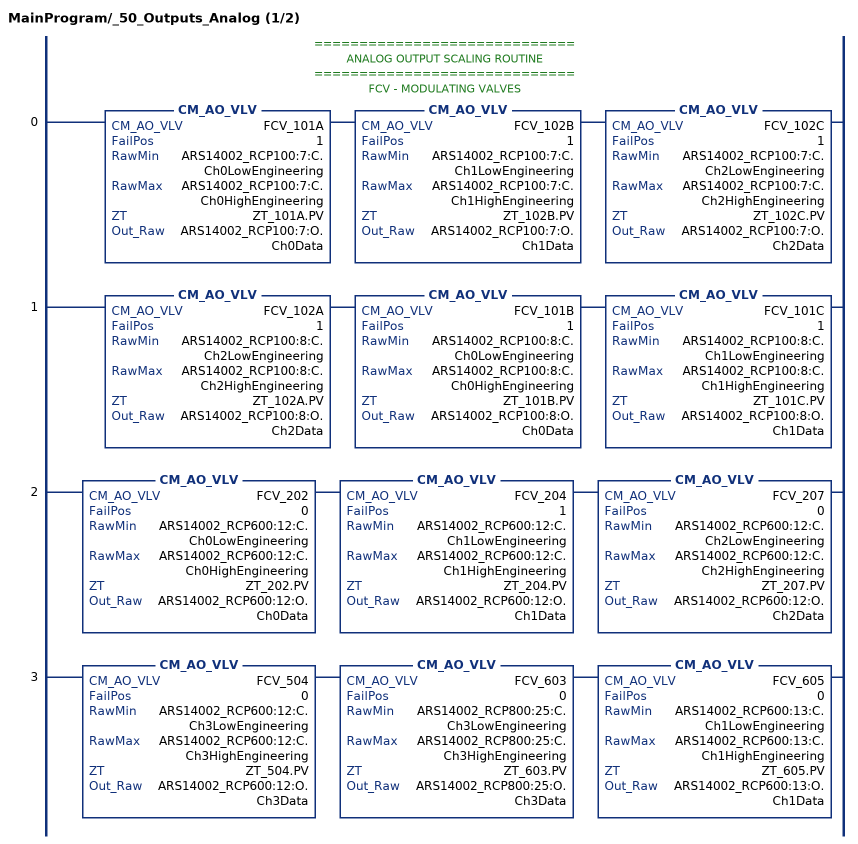
   // =============================
   // ANALOG OUTPUT SCALING ROUTINE
   // =============================
   // FCV - MODULATING VALVES
   0: CM_AO_VLV(FCV_101A,1,ARS14002_RCP100:7:C.Ch0LowEngineering,ARS14002_RCP100:7:C.Ch0HighEngineering,ZT_101A.PV,ARS14002_RCP100:7:O.Ch0Data)CM_AO_VLV(FCV_102B,1,ARS14002_RCP100:7:C.Ch1LowEngineering,ARS14002_RCP100:7:C.Ch1HighEngineering,ZT_102B.PV,ARS14002_RCP100:7:O.Ch1Data)CM_AO_VLV(FCV_102C,1,ARS14002_RCP100:7:C.Ch2LowEngineering,ARS14002_RCP100:7:C.Ch2HighEngineering,ZT_102C.PV,ARS14002_RCP100:7:O.Ch2Data);
   1: CM_AO_VLV(FCV_102A,1,ARS14002_RCP100:8:C.Ch2LowEngineering,ARS14002_RCP100:8:C.Ch2HighEngineering,ZT_102A.PV,ARS14002_RCP100:8:O.Ch2Data)CM_AO_VLV(FCV_101B,1,ARS14002_RCP100:8:C.Ch0LowEngineering,ARS14002_RCP100:8:C.Ch0HighEngineering,ZT_101B.PV,ARS14002_RCP100:8:O.Ch0Data)CM_AO_VLV(FCV_101C,1,ARS14002_RCP100:8:C.Ch1LowEngineering,ARS14002_RCP100:8:C.Ch1HighEngineering,ZT_101C.PV,ARS14002_RCP100:8:O.Ch1Data);
   2: CM_AO_VLV(FCV_202,0,ARS14002_RCP600:12:C.Ch0LowEngineering,ARS14002_RCP600:12:C.Ch0HighEngineering,ZT_202.PV,ARS14002_RCP600:12:O.Ch0Data)CM_AO_VLV(FCV_204,1,ARS14002_RCP600:12:C.Ch1LowEngineering,ARS14002_RCP600:12:C.Ch1HighEngineering,ZT_204.PV,ARS14002_RCP600:12:O.Ch1Data)CM_AO_VLV(FCV_207,0,ARS14002_RCP600:12:C.Ch2LowEngineering,ARS14002_RCP600:12:C.Ch2HighEngineering,ZT_207.PV,ARS14002_RCP600:12:O.Ch2Data);
   3: CM_AO_VLV(FCV_504,0,ARS14002_RCP600:12:C.Ch3LowEngineering,ARS14002_RCP600:12:C.Ch3HighEngineering,ZT_504.PV,ARS14002_RCP600:12:O.Ch3Data)CM_AO_VLV(FCV_603,0,ARS14002_RCP800:25:C.Ch3LowEngineering,ARS14002_RCP800:25:C.Ch3HighEngineering,ZT_603.PV,ARS14002_RCP800:25:O.Ch3Data)CM_AO_VLV(FCV_605,0,ARS14002_RCP600:13:C.Ch1LowEngineering,ARS14002_RCP600:13:C.Ch1HighEngineering,ZT_605.PV,ARS14002_RCP600:13:O.Ch1Data);
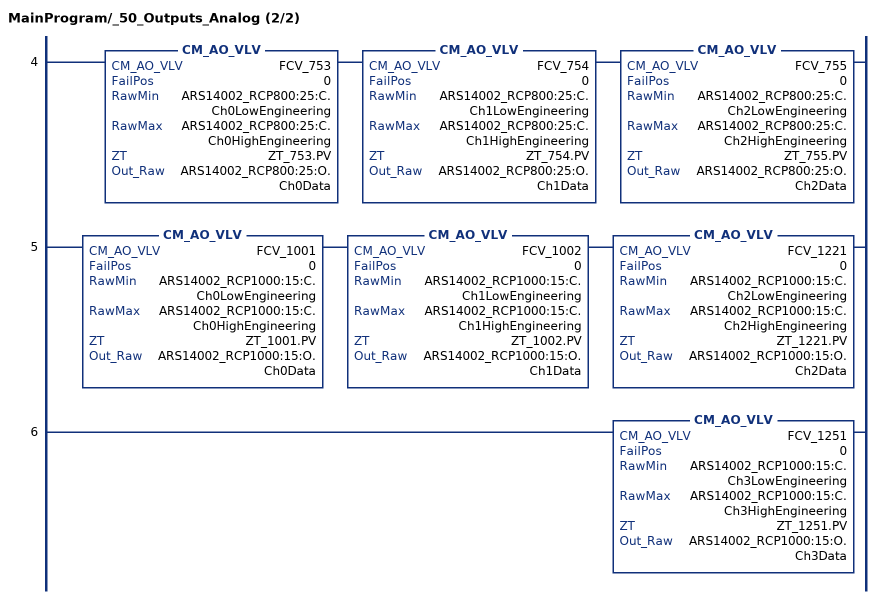
   4: CM_AO_VLV(FCV_753,0,ARS14002_RCP800:25:C.Ch0LowEngineering,ARS14002_RCP800:25:C.Ch0HighEngineering,ZT_753.PV,ARS14002_RCP800:25:O.Ch0Data)CM_AO_VLV(FCV_754,0,ARS14002_RCP800:25:C.Ch1LowEngineering,ARS14002_RCP800:25:C.Ch1HighEngineering,ZT_754.PV,ARS14002_RCP800:25:O.Ch1Data)CM_AO_VLV(FCV_755,0,ARS14002_RCP800:25:C.Ch2LowEngineering,ARS14002_RCP800:25:C.Ch2HighEngineering,ZT_755.PV,ARS14002_RCP800:25:O.Ch2Data);
   5: CM_AO_VLV(FCV_1001,0,ARS14002_RCP1000:15:C.Ch0LowEngineering,ARS14002_RCP1000:15:C.Ch0HighEngineering,ZT_1001.PV,ARS14002_RCP1000:15:O.Ch0Data)CM_AO_VLV(FCV_1002,0,ARS14002_RCP1000:15:C.Ch1LowEngineering,ARS14002_RCP1000:15:C.Ch1HighEngineering,ZT_1002.PV,ARS14002_RCP1000:15:O.Ch1Data)CM_AO_VLV(FCV_1221,0,ARS14002_RCP1000:15:C.Ch2LowEngineering,ARS14002_RCP1000:15:C.Ch2HighEngineering,ZT_1221.PV,ARS14002_RCP1000:15:O.Ch2Data);
   6: CM_AO_VLV(FCV_1251,0,ARS14002_RCP1000:15:C.Ch3LowEngineering,ARS14002_RCP1000:15:C.Ch3HighEngineering,ZT_1251.PV,ARS14002_RCP1000:15:O.Ch3Data);
END_ROUTINE
